{attribute 'GeneratedUsingTerminal: AT2026-0250-0019'}
{attribute addProperty BoxType "AT2026-0250-0019"}
{attribute addProperty Id "A_0077_AT2001_5250_0018_AT2001_5250AT2001_33A3DF1B80"}
{attribute addProperty CRC "2772908938"}
{attribute addProperty Size "80"}
TYPE A_0065_AT2026_0250_0019_AT2026_0250_A5473B8A EXTENDS AT2026_A7FEA1CF :
STRUCT
	{attribute addProperty Name "A_0077_AT2001_5250_0018_AT2001_5250"}
	{attribute addProperty PreviousPort "A_0065(AT2026-0250-0019) (AT2026-0250) : B"}
	A_0077_AT2001_5250_0018_AT2001_5250 : AT2001_33A3DF1B;
END_STRUCT
END_TYPE
